// TwinCAT 3 PLC project Untitled1
// ProgramVersion: 3.1.4023.0
// libraries:
//   Tc2_Standard, * (Beckhoff Automation GmbH)
//   Tc2_System, * (Beckhoff Automation GmbH)
//   Tc3_Module, * (Beckhoff Automation GmbH)
// project tree:
//   / PlcTask.TcTTO
//   POUs/ FB_ADD.TcPOU, MAIN.TcPOU, P_red.TcPOU
// real-time tasks:
//   TASK PlcTask: cycle T#10ms, priority 20, ADS port 350

CONFIGURATION Untitled1
    RESOURCE PLC ON TwinCAT3
        TASK PlcTask(INTERVAL := T#10ms, PRIORITY := 20);
        PROGRAM MAIN WITH PlcTask : MAIN;
    END_RESOURCE
END_CONFIGURATION

// ---- POUs/MAIN.TcPOU
PROGRAM MAIN
VAR
	a:INT;
	b:INT;
	c:INT;
	add1:FB_ADD;
	mux1:FB_MUX;
	ton1:Tc2_Standard.TON;
END_VAR

add1(in1:=a , in2:=b , out=>c );
ton1(IN:= , PT:=t#1s , Q=> , ET=> );

END_PROGRAM

// ---- POUs/FB_ADD.TcPOU
FUNCTION_BLOCK FB_ADD
VAR_INPUT
	in1,in2:INT;
END_VAR
VAR_OUTPUT
	out:INT;
END_VAR
VAR
END_VAR

out:=in1+in2;

END_FUNCTION_BLOCK

// ---- POUs/P_red.TcPOU
PROGRAM P_red
VAR
	a,b,c:INT;
END_VAR

c:=a*b;

END_PROGRAM
